FUNCTION_BLOCK FB_ReadAxisStatus
VAR_IN_OUT

AxisRef : AXIS_REF;

END_VAR

VAR_OUTPUT

AxisStatus : st_ReadAxis;

END_VAR
VAR	
END_VAR

AxisRef.ReadStatus();  
AxisStatus.Position			:= AxisRef.NcToPlc.ActPos;
AxisStatus.Velocity			:= AxisRef.NcToPlc.ActVelo;
AxisStatus.Acceleration		:= AxisRef.NcToPlc.ActAcc;
AxisStatus.Torque		    := AxisRef.NcToPlc.ActTorque;
//AxisStatus.Current			:= AxisRef.NcToPlc.ActTorque;
AxisStatus.ErrorID			:= AxisRef.NcToPlc.ErrorCode;

IF AxisRef.Status.ErrorStop THEN
	AxisStatus.eState := eAxis_ERRORSTOP;
ELSIF AxisRef.Status.Disabled THEN
	AxisStatus.eState := eAxis_DISABLED;
ELSIF AxisRef.Status.StandStill THEN
	AxisStatus.eState := eAxis_STANDSTILL;
ELSIF AxisRef.Status.Homing THEN
	AxisStatus.eState := eAxis_HOMING;
ELSIF AxisRef.Status.Stopping THEN
	AxisStatus.eState := eAxis_STOPPING;
ELSIF AxisRef.Status.DiscreteMotion THEN
	AxisStatus.eState := eAxis_DISCRETEMOTION;
ELSIF AxisRef.Status.ContinuousMotion THEN
	AxisStatus.eState := eAxis_CONTINOUSMOTION;
ELSIF AxisRef.Status.SynchronizedMotion THEN
	AxisStatus.eState := eAxis_SYNCHRONIZEDMOTION;
ELSE
	AxisStatus.eState := eAxis_UNDEFINED;
END_IF

END_FUNCTION_BLOCK

(* stored: Version 1.1.0.1, ProductVersion 3.1.4022.12
   POU FB_ReadAxisStatus: Id {df6ae7bd-09fc-46a8-8e9a-ef5fe5e1c5bf}, SpecialFunc None *)
